// TIA Portal V20 export
DATA_BLOCK "Enc"   // DB323
{ S7_Optimized_Access := 'TRUE' }
// stored: AutoNumber false, IsRetainMemResEnabled true, MemoryReserve 500, RetainMemoryReserve 500
   VAR RETAIN
      "1BCI1" : "TypeEncoder";   // encoder infeed scanner
      "1BCM1" : "TypeEncoder";   // encoder scanner
      "1BCO1" : "TypeEncoder";   // encoder outfeed scanner
      "8B1.B" : "TypeEncoder";   // light barrier measuring distance for the position of the scanner
      "8BC1.T" : "TypeEncoder";   // encoder adjustment top - normal drive
      "8BC1.L" : "TypeEncoder";   // encoder adjustment left - normal drive
      "8BC1.R" : "TypeEncoder";   // encoder adjustment right - normal drive
      "8U1.T" : "TypeEncoder";   // encoder adjustment top - linear drive
      "8U1.L" : "TypeEncoder";   // encoder adjustment left - linear drive
      "8U1.R" : "TypeEncoder";   // encoder adjustment right - linear drive
   END_VAR
BEGIN
   "1BCI1".ref := FALSE;
   "1BCI1".refMode := FALSE;
   "1BCI1".refRun := FALSE;
   "1BCI1".refOk := FALSE;
   "1BCI1".ready := TRUE;
   "1BCI1".posOk := TRUE;
   "1BCI1".notInPos := FALSE;
   "1BCI1".tarMin := TRUE;
   "1BCI1".tarMax := TRUE;
   "1BCI1".min := FALSE;
   "1BCI1".max := FALSE;
   "1BCI1".minTar := TRUE;
   "1BCI1".maxTar := TRUE;
   "1BCI1".sync := FALSE;
   "1BCI1".comOk := TRUE;
   "1BCI1".errOverflow := FALSE;
   "1BCI1".errRunCheck := FALSE;
   "1BCI1".errLim := FALSE;
   "1BCI1".errCom := FALSE;
   "1BCI1".err := FALSE;
   "1BCI1".errOffDel := TRUE;
   "1BCI1".dirUp := FALSE;
   "1BCI1".dirDn := TRUE;
   "1BCI1".errNr := 0;
   "1BCI1".encAct := 0;
   "1BCI1".resetPos := 0.0;
   "1BCI1".calOffset := 0.0;
   "1BCI1".calGain := 0.0005025126;
   "1BCI1".refPos := 0.0;
   "1BCI1".calP1Inc := 0;
   "1BCI1".calP1Mm := 0.0;
   "1BCI1".calP2Inc := 0;
   "1BCI1".calP2Mm := 0.0;
   "1BCI1".limMin := 0.0;
   "1BCI1".limMax := 0.0;
   "1BCI1".tar := 10.0;
   "1BCI1".act := 0.0;
   "1BCI1".offset := 0.0;
   "1BCI1".deltaInc := 0;
   "1BCI1".delta := 11.31196;
   "1BCI1".tarMinPos := 10.0;
   "1BCI1".tarMaxPos := -10.0;
   "1BCI1".minPos := 0.0;
   "1BCI1".maxPos := 0.0;
   "1BCI1".gPos := 0.0;
   "1BCI1".ePos := 0.0;
   "1BCI1".sPos := 0.0;
   "1BCI1".speed := 16#7FBF_FFFF;
   "1BCI1"."name" := WSTRING#'35BC11';
   "1BCI1".description := WSTRING#'Encoder Zuteiler Anschlag - Zubringung';
   "1BCM1".ref := FALSE;
   "1BCM1".refMode := FALSE;
   "1BCM1".refRun := FALSE;
   "1BCM1".refOk := FALSE;
   "1BCM1".ready := FALSE;
   "1BCM1".posOk := TRUE;
   "1BCM1".notInPos := FALSE;
   "1BCM1".tarMin := TRUE;
   "1BCM1".tarMax := TRUE;
   "1BCM1".min := FALSE;
   "1BCM1".max := FALSE;
   "1BCM1".minTar := TRUE;
   "1BCM1".maxTar := TRUE;
   "1BCM1".sync := FALSE;
   "1BCM1".comOk := FALSE;
   "1BCM1".errOverflow := FALSE;
   "1BCM1".errRunCheck := FALSE;
   "1BCM1".errLim := TRUE;
   "1BCM1".errCom := TRUE;
   "1BCM1".err := FALSE;
   "1BCM1".errOffDel := TRUE;
   "1BCM1".dirUp := FALSE;
   "1BCM1".dirDn := FALSE;
   "1BCM1".errNr := 112;
   "1BCM1".encAct := 0;
   "1BCM1".resetPos := 0.0;
   "1BCM1".calOffset := 0.0;
   "1BCM1".calGain := 0.0;
   "1BCM1".refPos := 0.0;
   "1BCM1".calP1Inc := 0;
   "1BCM1".calP1Mm := 0.0;
   "1BCM1".calP2Inc := 0;
   "1BCM1".calP2Mm := 0.0;
   "1BCM1".limMin := -50.0;
   "1BCM1".limMax := 50.0;
   "1BCM1".tar := 10.0;
   "1BCM1".act := 0.0;
   "1BCM1".offset := 0.0;
   "1BCM1".deltaInc := 0;
   "1BCM1".delta := 11.31196;
   "1BCM1".tarMinPos := 10.0;
   "1BCM1".tarMaxPos := -10.0;
   "1BCM1".minPos := 0.0;
   "1BCM1".maxPos := 0.0;
   "1BCM1".gPos := 0.0;
   "1BCM1".ePos := 0.0;
   "1BCM1".sPos := 0.0;
   "1BCM1".speed := 0.0;
   "1BCM1"."name" := WSTRING#'35BC11';
   "1BCM1".description := WSTRING#'Encoder Zuteiler Anschlag - Zubringung';
   "1BCO1".ref := FALSE;
   "1BCO1".refMode := FALSE;
   "1BCO1".refRun := FALSE;
   "1BCO1".refOk := FALSE;
   "1BCO1".ready := FALSE;
   "1BCO1".posOk := TRUE;
   "1BCO1".notInPos := FALSE;
   "1BCO1".tarMin := TRUE;
   "1BCO1".tarMax := TRUE;
   "1BCO1".min := FALSE;
   "1BCO1".max := FALSE;
   "1BCO1".minTar := TRUE;
   "1BCO1".maxTar := TRUE;
   "1BCO1".sync := FALSE;
   "1BCO1".comOk := FALSE;
   "1BCO1".errOverflow := FALSE;
   "1BCO1".errRunCheck := FALSE;
   "1BCO1".errLim := TRUE;
   "1BCO1".errCom := TRUE;
   "1BCO1".err := FALSE;
   "1BCO1".errOffDel := TRUE;
   "1BCO1".dirUp := FALSE;
   "1BCO1".dirDn := FALSE;
   "1BCO1".errNr := 112;
   "1BCO1".encAct := 0;
   "1BCO1".resetPos := 0.0;
   "1BCO1".calOffset := 0.0;
   "1BCO1".calGain := 0.0;
   "1BCO1".refPos := 0.0;
   "1BCO1".calP1Inc := 0;
   "1BCO1".calP1Mm := 0.0;
   "1BCO1".calP2Inc := 0;
   "1BCO1".calP2Mm := 0.0;
   "1BCO1".limMin := -50.0;
   "1BCO1".limMax := 50.0;
   "1BCO1".tar := 10.0;
   "1BCO1".act := 0.0;
   "1BCO1".offset := 0.0;
   "1BCO1".deltaInc := 0;
   "1BCO1".delta := 11.31196;
   "1BCO1".tarMinPos := 10.0;
   "1BCO1".tarMaxPos := -10.0;
   "1BCO1".minPos := 0.0;
   "1BCO1".maxPos := 0.0;
   "1BCO1".gPos := 0.0;
   "1BCO1".ePos := 0.0;
   "1BCO1".sPos := 0.0;
   "1BCO1".speed := 0.0;
   "1BCO1"."name" := WSTRING#'35BC11';
   "1BCO1".description := WSTRING#'Encoder Zuteiler Anschlag - Zubringung';
   "8B1.B".ref := FALSE;
   "8B1.B".refMode := FALSE;
   "8B1.B".refRun := FALSE;
   "8B1.B".refOk := TRUE;
   "8B1.B".ready := FALSE;
   "8B1.B".posOk := FALSE;
   "8B1.B".notInPos := FALSE;
   "8B1.B".tarMin := FALSE;
   "8B1.B".tarMax := FALSE;
   "8B1.B".min := FALSE;
   "8B1.B".max := FALSE;
   "8B1.B".minTar := FALSE;
   "8B1.B".maxTar := FALSE;
   "8B1.B".sync := FALSE;
   "8B1.B".comOk := FALSE;
   "8B1.B".errOverflow := FALSE;
   "8B1.B".errRunCheck := FALSE;
   "8B1.B".errLim := FALSE;
   "8B1.B".errCom := FALSE;
   "8B1.B".err := FALSE;
   "8B1.B".errOffDel := FALSE;
   "8B1.B".dirUp := FALSE;
   "8B1.B".dirDn := FALSE;
   "8B1.B".errNr := 0;
   "8B1.B".encAct := -2360;
   "8B1.B".resetPos := 0.0;
   "8B1.B".calOffset := 0.0;
   "8B1.B".calGain := 1.0;
   "8B1.B".refPos := 0.0;
   "8B1.B".calP1Inc := 0;
   "8B1.B".calP1Mm := 0.0;
   "8B1.B".calP2Inc := 0;
   "8B1.B".calP2Mm := 0.0;
   "8B1.B".limMin := -505.0;
   "8B1.B".limMax := 505.0;
   "8B1.B".tar := 60.0;
   "8B1.B".act := -236.0;
   "8B1.B".offset := 0.0;
   "8B1.B".deltaInc := 0;
   "8B1.B".delta := 0.0;
   "8B1.B".tarMinPos := -500.0;
   "8B1.B".tarMaxPos := 500.0;
   "8B1.B".minPos := -500.0;
   "8B1.B".maxPos := 500.0;
   "8B1.B".gPos := 0.0;
   "8B1.B".ePos := 0.0;
   "8B1.B".sPos := 0.0;
   "8B1.B".speed := 0.0;
   "8B1.B"."name" := WSTRING#'';
   "8B1.B".description := WSTRING#'';
   "8BC1.T".ref := FALSE;
   "8BC1.T".refMode := TRUE;
   "8BC1.T".refRun := FALSE;
   "8BC1.T".refOk := TRUE;
   "8BC1.T".ready := TRUE;
   "8BC1.T".posOk := FALSE;
   "8BC1.T".notInPos := FALSE;
   "8BC1.T".tarMin := FALSE;
   "8BC1.T".tarMax := FALSE;
   "8BC1.T".min := FALSE;
   "8BC1.T".max := FALSE;
   "8BC1.T".minTar := TRUE;
   "8BC1.T".maxTar := FALSE;
   "8BC1.T".sync := FALSE;
   "8BC1.T".comOk := TRUE;
   "8BC1.T".errOverflow := FALSE;
   "8BC1.T".errRunCheck := FALSE;
   "8BC1.T".errLim := TRUE;
   "8BC1.T".errCom := FALSE;
   "8BC1.T".err := TRUE;
   "8BC1.T".errOffDel := TRUE;
   "8BC1.T".dirUp := TRUE;
   "8BC1.T".dirDn := FALSE;
   "8BC1.T".errNr := 1;
   "8BC1.T".encAct := 1563;
   "8BC1.T".resetPos := 52.98273;
   "8BC1.T".calOffset := 0.0;
   "8BC1.T".calGain := -0.0275;
   "8BC1.T".refPos := 10.0;
   "8BC1.T".calP1Inc := 0;
   "8BC1.T".calP1Mm := 0.0;
   "8BC1.T".calP2Inc := 0;
   "8BC1.T".calP2Mm := 0.0;
   "8BC1.T".limMin := 5.0;
   "8BC1.T".limMax := 215.0;
   "8BC1.T".tar := 12.0;
   "8BC1.T".act := -32.98265;
   "8BC1.T".offset := 0.0;
   "8BC1.T".deltaInc := 0;
   "8BC1.T".delta := 0.0;
   "8BC1.T".tarMinPos := 10.0;
   "8BC1.T".tarMaxPos := 210.0;
   "8BC1.T".minPos := 10.0;
   "8BC1.T".maxPos := 210.0;
   "8BC1.T".gPos := 0.0;
   "8BC1.T".ePos := 0.0;
   "8BC1.T".sPos := 0.0;
   "8BC1.T".speed := 16#7FBF_FFFF;
   "8BC1.T"."name" := WSTRING#'35BC11';
   "8BC1.T".description := WSTRING#'Encoder Zuteiler Anschlag - Zubringung';
   "8BC1.L".ref := FALSE;
   "8BC1.L".refMode := TRUE;
   "8BC1.L".refRun := FALSE;
   "8BC1.L".refOk := TRUE;
   "8BC1.L".ready := TRUE;
   "8BC1.L".posOk := TRUE;
   "8BC1.L".notInPos := FALSE;
   "8BC1.L".tarMin := FALSE;
   "8BC1.L".tarMax := FALSE;
   "8BC1.L".min := FALSE;
   "8BC1.L".max := FALSE;
   "8BC1.L".minTar := FALSE;
   "8BC1.L".maxTar := FALSE;
   "8BC1.L".sync := FALSE;
   "8BC1.L".comOk := TRUE;
   "8BC1.L".errOverflow := FALSE;
   "8BC1.L".errRunCheck := FALSE;
   "8BC1.L".errLim := FALSE;
   "8BC1.L".errCom := FALSE;
   "8BC1.L".err := FALSE;
   "8BC1.L".errOffDel := FALSE;
   "8BC1.L".dirUp := TRUE;
   "8BC1.L".dirDn := FALSE;
   "8BC1.L".errNr := 0;
   "8BC1.L".encAct := 638;
   "8BC1.L".resetPos := 9.972851;
   "8BC1.L".calOffset := 0.0;
   "8BC1.L".calGain := -0.0275;
   "8BC1.L".refPos := 10.0;
   "8BC1.L".calP1Inc := 0;
   "8BC1.L".calP1Mm := 0.0;
   "8BC1.L".calP2Inc := 0;
   "8BC1.L".calP2Mm := 0.0;
   "8BC1.L".limMin := 5.0;
   "8BC1.L".limMax := 215.0;
   "8BC1.L".tar := 87.5;
   "8BC1.L".act := 87.52025;
   "8BC1.L".offset := 0.0;
   "8BC1.L".deltaInc := 0;
   "8BC1.L".delta := 0.0;
   "8BC1.L".tarMinPos := 10.0;
   "8BC1.L".tarMaxPos := 210.0;
   "8BC1.L".minPos := 10.0;
   "8BC1.L".maxPos := 210.0;
   "8BC1.L".gPos := 0.0;
   "8BC1.L".ePos := 0.0;
   "8BC1.L".sPos := 0.0;
   "8BC1.L".speed := 16#7FBF_FFFF;
   "8BC1.L"."name" := WSTRING#'35BC11';
   "8BC1.L".description := WSTRING#'Encoder Zuteiler Anschlag - Zubringung';
   "8BC1.R".ref := FALSE;
   "8BC1.R".refMode := TRUE;
   "8BC1.R".refRun := FALSE;
   "8BC1.R".refOk := TRUE;
   "8BC1.R".ready := TRUE;
   "8BC1.R".posOk := TRUE;
   "8BC1.R".notInPos := FALSE;
   "8BC1.R".tarMin := FALSE;
   "8BC1.R".tarMax := FALSE;
   "8BC1.R".min := FALSE;
   "8BC1.R".max := FALSE;
   "8BC1.R".minTar := FALSE;
   "8BC1.R".maxTar := FALSE;
   "8BC1.R".sync := FALSE;
   "8BC1.R".comOk := TRUE;
   "8BC1.R".errOverflow := FALSE;
   "8BC1.R".errRunCheck := FALSE;
   "8BC1.R".errLim := FALSE;
   "8BC1.R".errCom := FALSE;
   "8BC1.R".err := FALSE;
   "8BC1.R".errOffDel := FALSE;
   "8BC1.R".dirUp := TRUE;
   "8BC1.R".dirDn := FALSE;
   "8BC1.R".errNr := 0;
   "8BC1.R".encAct := 636;
   "8BC1.R".resetPos := 10.00027;
   "8BC1.R".calOffset := 0.0;
   "8BC1.R".calGain := -0.0275;
   "8BC1.R".refPos := 10.0;
   "8BC1.R".calP1Inc := 0;
   "8BC1.R".calP1Mm := 0.0;
   "8BC1.R".calP2Inc := 0;
   "8BC1.R".calP2Mm := 0.0;
   "8BC1.R".limMin := 5.0;
   "8BC1.R".limMax := 215.0;
   "8BC1.R".tar := 82.6;
   "8BC1.R".act := 82.62568;
   "8BC1.R".offset := 0.0;
   "8BC1.R".deltaInc := 0;
   "8BC1.R".delta := 0.0;
   "8BC1.R".tarMinPos := 10.0;
   "8BC1.R".tarMaxPos := 210.0;
   "8BC1.R".minPos := 10.0;
   "8BC1.R".maxPos := 210.0;
   "8BC1.R".gPos := 0.0;
   "8BC1.R".ePos := 0.0;
   "8BC1.R".sPos := 0.0;
   "8BC1.R".speed := 16#7FBF_FFFF;
   "8BC1.R"."name" := WSTRING#'35BC11';
   "8BC1.R".description := WSTRING#'Encoder Zuteiler Anschlag - Zubringung';
   "8U1.T".ref := TRUE;
   "8U1.T".refMode := TRUE;
   "8U1.T".refRun := FALSE;
   "8U1.T".refOk := FALSE;
   "8U1.T".ready := FALSE;
   "8U1.T".posOk := FALSE;
   "8U1.T".notInPos := FALSE;
   "8U1.T".tarMin := TRUE;
   "8U1.T".tarMax := TRUE;
   "8U1.T".min := FALSE;
   "8U1.T".max := FALSE;
   "8U1.T".minTar := TRUE;
   "8U1.T".maxTar := TRUE;
   "8U1.T".sync := FALSE;
   "8U1.T".comOk := FALSE;
   "8U1.T".errOverflow := FALSE;
   "8U1.T".errRunCheck := FALSE;
   "8U1.T".errLim := TRUE;
   "8U1.T".errCom := TRUE;
   "8U1.T".err := FALSE;
   "8U1.T".errOffDel := TRUE;
   "8U1.T".dirUp := FALSE;
   "8U1.T".dirDn := FALSE;
   "8U1.T".errNr := 112;
   "8U1.T".encAct := 0;
   "8U1.T".resetPos := 0.0;
   "8U1.T".calOffset := 0.0;
   "8U1.T".calGain := 1.0;
   "8U1.T".refPos := 0.0;
   "8U1.T".calP1Inc := 0;
   "8U1.T".calP1Mm := 0.0;
   "8U1.T".calP2Inc := 0;
   "8U1.T".calP2Mm := 0.0;
   "8U1.T".limMin := -5.0;
   "8U1.T".limMax := 155.0;
   "8U1.T".tar := 42.0;
   "8U1.T".act := 0.0;
   "8U1.T".offset := 0.0;
   "8U1.T".deltaInc := 0;
   "8U1.T".delta := 0.0;
   "8U1.T".tarMinPos := 0.0;
   "8U1.T".tarMaxPos := 150.0;
   "8U1.T".minPos := 0.0;
   "8U1.T".maxPos := 150.0;
   "8U1.T".gPos := 0.0;
   "8U1.T".ePos := 0.0;
   "8U1.T".sPos := 0.0;
   "8U1.T".speed := 0.0;
   "8U1.T"."name" := WSTRING#'35BC11';
   "8U1.T".description := WSTRING#'Encoder Zuteiler Anschlag - Zubringung';
   "8U1.L".ref := TRUE;
   "8U1.L".refMode := TRUE;
   "8U1.L".refRun := FALSE;
   "8U1.L".refOk := FALSE;
   "8U1.L".ready := FALSE;
   "8U1.L".posOk := FALSE;
   "8U1.L".notInPos := FALSE;
   "8U1.L".tarMin := TRUE;
   "8U1.L".tarMax := TRUE;
   "8U1.L".min := FALSE;
   "8U1.L".max := FALSE;
   "8U1.L".minTar := TRUE;
   "8U1.L".maxTar := TRUE;
   "8U1.L".sync := FALSE;
   "8U1.L".comOk := FALSE;
   "8U1.L".errOverflow := FALSE;
   "8U1.L".errRunCheck := FALSE;
   "8U1.L".errLim := TRUE;
   "8U1.L".errCom := TRUE;
   "8U1.L".err := FALSE;
   "8U1.L".errOffDel := TRUE;
   "8U1.L".dirUp := FALSE;
   "8U1.L".dirDn := FALSE;
   "8U1.L".errNr := 112;
   "8U1.L".encAct := 0;
   "8U1.L".resetPos := 0.0;
   "8U1.L".calOffset := 0.0;
   "8U1.L".calGain := 1.0;
   "8U1.L".refPos := 0.0;
   "8U1.L".calP1Inc := 0;
   "8U1.L".calP1Mm := 0.0;
   "8U1.L".calP2Inc := 0;
   "8U1.L".calP2Mm := 0.0;
   "8U1.L".limMin := -5.0;
   "8U1.L".limMax := 155.0;
   "8U1.L".tar := 82.5;
   "8U1.L".act := 0.0;
   "8U1.L".offset := 0.0;
   "8U1.L".deltaInc := 0;
   "8U1.L".delta := 0.0;
   "8U1.L".tarMinPos := 0.0;
   "8U1.L".tarMaxPos := 150.0;
   "8U1.L".minPos := 0.0;
   "8U1.L".maxPos := 150.0;
   "8U1.L".gPos := 0.0;
   "8U1.L".ePos := 0.0;
   "8U1.L".sPos := 0.0;
   "8U1.L".speed := 0.0;
   "8U1.L"."name" := WSTRING#'35BC11';
   "8U1.L".description := WSTRING#'Encoder Zuteiler Anschlag - Zubringung';
   "8U1.R".ref := TRUE;
   "8U1.R".refMode := TRUE;
   "8U1.R".refRun := FALSE;
   "8U1.R".refOk := FALSE;
   "8U1.R".ready := FALSE;
   "8U1.R".posOk := FALSE;
   "8U1.R".notInPos := FALSE;
   "8U1.R".tarMin := TRUE;
   "8U1.R".tarMax := TRUE;
   "8U1.R".min := FALSE;
   "8U1.R".max := FALSE;
   "8U1.R".minTar := TRUE;
   "8U1.R".maxTar := TRUE;
   "8U1.R".sync := FALSE;
   "8U1.R".comOk := FALSE;
   "8U1.R".errOverflow := FALSE;
   "8U1.R".errRunCheck := FALSE;
   "8U1.R".errLim := TRUE;
   "8U1.R".errCom := TRUE;
   "8U1.R".err := FALSE;
   "8U1.R".errOffDel := TRUE;
   "8U1.R".dirUp := FALSE;
   "8U1.R".dirDn := FALSE;
   "8U1.R".errNr := 112;
   "8U1.R".encAct := 0;
   "8U1.R".resetPos := 0.0;
   "8U1.R".calOffset := 0.0;
   "8U1.R".calGain := 1.0;
   "8U1.R".refPos := 0.0;
   "8U1.R".calP1Inc := 0;
   "8U1.R".calP1Mm := 0.0;
   "8U1.R".calP2Inc := 0;
   "8U1.R".calP2Mm := 0.0;
   "8U1.R".limMin := -5.0;
   "8U1.R".limMax := 155.0;
   "8U1.R".tar := 82.5;
   "8U1.R".act := 0.0;
   "8U1.R".offset := 0.0;
   "8U1.R".deltaInc := 0;
   "8U1.R".delta := 0.0;
   "8U1.R".tarMinPos := 0.0;
   "8U1.R".tarMaxPos := 150.0;
   "8U1.R".minPos := 0.0;
   "8U1.R".maxPos := 150.0;
   "8U1.R".gPos := 0.0;
   "8U1.R".ePos := 0.0;
   "8U1.R".sPos := 0.0;
   "8U1.R".speed := 0.0;
   "8U1.R"."name" := WSTRING#'35BC11';
   "8U1.R".description := WSTRING#'Encoder Zuteiler Anschlag - Zubringung';
END_DATA_BLOCK
